// Mitsubishi GX Works2 project: 231002-001- exercicios-2   PLC: Q03UDV

// task Task_01 (event TRUE, interval 0, priority 31): POU_01

PROGRAM POU_01
VAR
  CTD_1 : CTD;
  CTU_1 : CTU;
  meuc : CTU;
END_VAR
(* structured ladder/FBD written out as ST: instructions are called as NAME(EN, inputs, outputs); _pN, _eN, _tN stand for wires *)
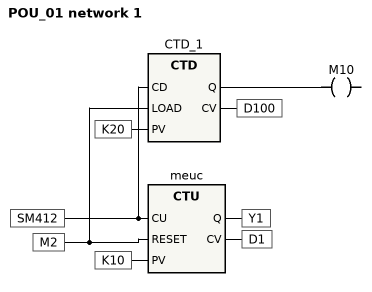
(* network 1 *)
CTD_1(CD := SM412, LOAD := M2, PV := K20, CV => D100);
M10 := CTD_1.Q;
meuc(CU := SM412, RESET := M2, PV := K10, Q => Y1, CV => D1);
END_PROGRAM
